FUNCTION Pow3 : LREAL
VAR_INPUT
	number : LREAL;
END_VAR

Pow3 := number * number * number;

END_FUNCTION

(* stored: Version 1.1.0.1
   POU Pow3: Id {6c6a1f87-6dfb-0c65-39e0-c1d43287ffe2}, SpecialFunc None *)
